{attribute 'linkalways'} 
{attribute 'no_explicit_call' := 'This FB is a CLASS and must be accessed using methods or properties'}
{attribute 'enable_dynamic_creation'}
FUNCTION_BLOCK Node_F_VN_AppendToContainer_INT EXTENDS Node
VAR
    nElement : _INT(0);
    ipContainer : _ITcVnContainer;
    hrPrev : _HRESULT(S_OK);
	hresult : _HRESULT(S_OK);
END_VAR

METHOD PUBLIC  Clone : I_Node
VAR
	pNode : POINTER TO Node_F_VN_AppendToContainer_INT;
END_VAR
pNode := __NEW(Node_F_VN_AppendToContainer_INT);
Clone := pNode^;
END_METHOD

METHOD FB_init : BOOL
VAR_INPUT
	bInitRetains : BOOL; // if TRUE, the retain variables are initialized (warm start / cold start)
	bInCopyCode : BOOL;  // if TRUE, the instance afterwards gets moved into the copy code (online change)
END_VAR
AddInput('nElement', nElement);
AddInput('ipContainer', ipContainer);
AddInput('hrPrev', hrPrev);
AddOutput('ipContainer', ipContainer);
AddOutput('hresult',hresult);
END_METHOD

METHOD PROTECTED OnExecute : HRESULT
hresult.Value := F_VN_AppendToContainer_INT(
    nElement := nElement.Value,
	ipContainer := ipContainer.Value,
	hrPrev:= hrPrev.Value);
END_METHOD

END_FUNCTION_BLOCK

(* stored: Version 1.1.0.1, ProductVersion 3.1.4024.13
   POU Node_F_VN_AppendToContainer_INT: Id {52c9c464-cfea-00b1-14d9-63e07123ab45}, SpecialFunc None
   Folder Constructor: Id {1888b2b2-a46c-0c4e-198e-c7914649bfe6}
   Method Clone: Id {2a43f38a-5d5e-01c2-22d1-2790dab27bb2}
   Method FB_init: Id {7a40b9f9-db68-0625-3bec-41c446a793c3}
   Method OnExecute: Id {1db72227-2dd7-0271-031e-f47e157866f5} *)
